// TwinCAT 3 PLC project Untitled1
// ProgramVersion: 3.1.4023.0
// libraries:
//   Tc2_Standard, * (Beckhoff Automation GmbH)
//   Tc2_System, * (Beckhoff Automation GmbH)
//   Tc2_Utilities, * (Beckhoff Automation GmbH)
//   Tc3_Module, * (Beckhoff Automation GmbH)
// project tree:
//   / PlcTask.TcTTO
//   POUs/ MAIN.TcPOU
// real-time tasks:
//   TASK PlcTask: cycle T#10ms, priority 20, ADS port 350

CONFIGURATION Untitled1
    RESOURCE PLC ON TwinCAT3
        TASK PlcTask(INTERVAL := T#10ms, PRIORITY := 20);
        PROGRAM MAIN WITH PlcTask : MAIN;
    END_RESOURCE
END_CONFIGURATION

// ---- POUs/MAIN.TcPOU
PROGRAM MAIN
VAR
	fbRand : DRAND;
	lrRandomValue : LREAL;
	rTemp : REAL;
	rAlarmHigh : REAL := 40.0;
	rAlarmLow : REAL := -40.0;
	rWarningHigh : REAL := 30.0;
	rWarningLow : REAL := -30.0;
	rVariableOffset: REAL;
END_VAR

fbRand(Seed := 0, Num => lrRandomValue);
rTemp := (LREAL_TO_REAL(lrRandomValue) * 100.0) - 50.0;

END_PROGRAM
